INTERFACE I_Channel EXTENDS I_Object

PROPERTY PUBLIC P_ID : String(25)
GET
END_GET
END_PROPERTY

PROPERTY PUBLIC P_MappingStatus : EPlcMappingStatus
GET
END_GET
END_PROPERTY

END_INTERFACE

(* stored: Version 1.1.0.1
   Itf I_Channel: Id {1b297b6b-809c-0abd-3ee4-a73d9efd4868}
   Property P_ID: Id {84f9e729-2b72-054c-28a1-316d6cb797db}
   Get Get: Id {90a42a60-8a97-06d5-2237-4e83f6005a9c}
   Property P_MappingStatus: Id {422b6820-34d0-001c-08fb-4d532a6b4877}
   Get Get: Id {6df90bef-98f8-013a-0e1f-b6e2b5def842} *)
